// SIMATIC S7-200 project (STEP 7-Micro/WIN), CPU 224 REL 02.01

ORGANIZATION_BLOCK MAIN:OB1
TITLE=PROGRAM COMMENTS
BEGIN
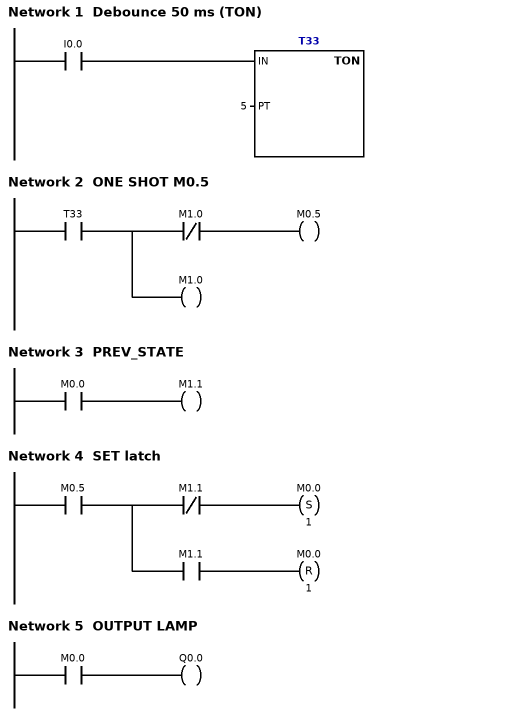
Network 1 // Debounce 50 ms (TON)
LD     I0.0
TON    T33, 5
Network 2 // ONE SHOT M0.5
LD     T33
LPS
AN     M1.0
=      M0.5
LPP
=      M1.0
Network 3 // PREV_STATE
LD     M0.0
=      M1.1
Network 4 // SET latch
LD     M0.5
LPS
AN     M1.1
S      M0.0, 1
LPP
A      M1.1
R      M0.0, 1
Network 5 // OUTPUT LAMP
LD     M0.0
=      Q0.0
END_ORGANIZATION_BLOCK
